Universal Robots PolyScope program: reciprocal_p1_3.urp

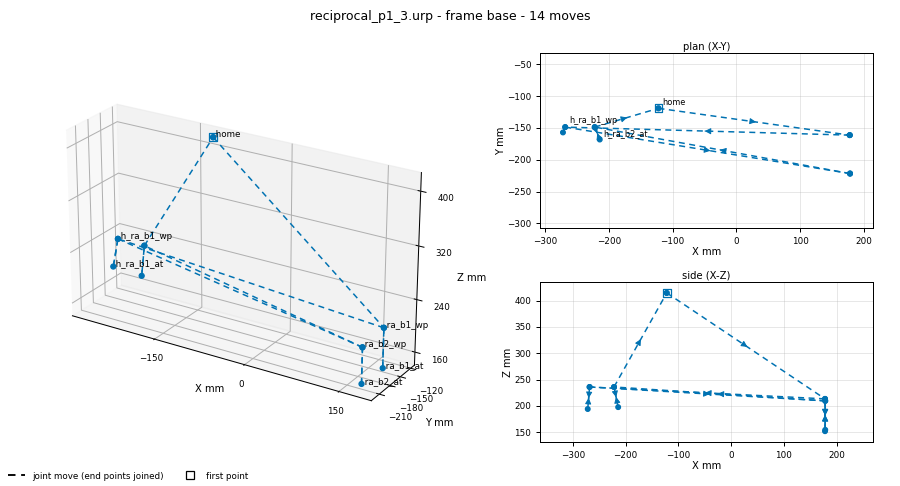
[picture p0: tool path of reciprocal_p1_3.urp in frame base, 14 of 14 moves have a stored position in this frame; points joined in program order, loops and branches not executed]
Program reciprocal_p1_3 (installation=default directory=/programs/usbdisk/ITER createdIn=5.3.1.64192 lastSavedIn=5.3.1.64192 robotSerialNumber=20195300365)
Calibrated DH parameters: a=[-0.000093, -0.190649, -0.212673, 0.000091, -0.000205, 0]; d=[0.151591, 44.061648, -42.488068, -1.442789, 0.085322, 0.091911]; alpha=[1.570082, -0.003447, 0.007513, 1.572293, -1.571904, 0]; deltaTheta=[0, -0.672656, 0.728185, -0.055522, 0.000005, 0]
Robot Program (runOnlyOnce=false)
  URCap Gripper Activate (Robotiq_Grippers, Robotiq Inc.) dataModel(ResetAndActivateKey=false)
  URCap Gripper (Robotiq_Grippers, Robotiq Inc.) dataModel(position=50.0, force=100.0, speed=100.0, positionInDouble=50.0, forceInDouble=100.0, speedInDouble=100.0, slaveIds=[9], blocking=true)
  MoveJ speed 60 deg/s, acceleration 80 deg/s^2 (useActiveTCP=true) feature=Base
    Waypoint home: TCP in base x=-122.15 y=-119.32 z=414.454 mm, rx=2.2563 ry=2.1459 rz=-0.0481 rad; joints [-85.681, -56.776, -79.802, -131.025, 89.944, -262.833] deg
  Folder Roof_A
    MoveJ speed 60 deg/s, acceleration 80 deg/s^2 (useActiveTCP=true) feature=Base
      Waypoint ra_b1_wp: TCP in base x=178.147 y=-161.416 z=213.493 mm, rx=2.2107 ry=2.1864 rz=-0.0129 rad; joints [-8.931, -69.528, -131.792, -67.419, 88.9, -187.899] deg
      Waypoint ra_b1_at: TCP in base x=178.14 y=-161.425 z=152.15 mm, rx=2.2108 ry=2.1863 rz=-0.013 rad; joints [-8.971, -81.208, -143.947, -43.587, 88.771, -187.8] deg
      URCap Gripper (Robotiq_Grippers, Robotiq Inc.) dataModel(position=100.0, force=100.0, speed=100.0, positionInDouble=100.0, forceInDouble=100.0, speedInDouble=100.0, slaveIds=[9], blocking=true)
      Waypoint ra_b1_wp: TCP in base x=178.147 y=-161.416 z=213.493 mm, rx=2.2107 ry=2.1864 rz=-0.0129 rad; joints [-8.931, -69.528, -131.792, -67.419, 88.9, -187.899] deg
      Waypoint h_ra_b1_wp: TCP in base x=-268.55 y=-148.787 z=236.04 mm, rx=2.7608 ry=-0.1306 rz=0.0749 rad; joints [-131.096, -88.368, -118.927, -47.1, 105.838, -213.026] deg
      Waypoint h_ra_b1_at: TCP in base x=-272.048 y=-157.193 z=194.251 mm, rx=2.7928 ry=-0.086 rz=0.1068 rad; joints [-130.55, -96.287, -122.586, -37.872, 105.802, -214.66] deg
      URCap Gripper (Robotiq_Grippers, Robotiq Inc.) dataModel(position=50.0, force=100.0, speed=100.0, positionInDouble=50.0, forceInDouble=100.0, speedInDouble=100.0, slaveIds=[9], blocking=true)
      Waypoint h_ra_b1_wp: TCP in base x=-268.55 y=-148.787 z=236.04 mm, rx=2.7608 ry=-0.1306 rz=0.0749 rad; joints [-131.096, -88.368, -118.927, -47.1, 105.838, -213.026] deg
    MoveJ speed 60 deg/s, acceleration 80 deg/s^2 (useActiveTCP=true) feature=Base
      Waypoint ra_b2_wp: TCP in base x=178.587 y=-221.707 z=209.682 mm, rx=2.2093 ry=2.1872 rz=-0.0611 rad; joints [-23.097, -83.646, -122.705, -62.748, 87.545, -202.118] deg
      Waypoint ra_b2_at: TCP in base x=178.563 y=-221.705 z=154.679 mm, rx=2.2094 ry=2.1872 rz=-0.0612 rad; joints [-23.123, -93.044, -131.897, -44.166, 87.443, -202.046] deg
      URCap Gripper (Robotiq_Grippers, Robotiq Inc.) dataModel(position=100.0, force=100.0, speed=100.0, positionInDouble=100.0, forceInDouble=100.0, speedInDouble=100.0, slaveIds=[9], blocking=true)
      Waypoint ra_b2_wp: TCP in base x=178.587 y=-221.707 z=209.682 mm, rx=2.2093 ry=2.1872 rz=-0.0611 rad; joints [-23.097, -83.646, -122.705, -62.748, 87.545, -202.118] deg
      Waypoint h_ra_b2_wp: TCP in base x=-222.173 y=-148.778 z=236.048 mm, rx=2.7617 ry=-0.0717 rz=0.0011 rad; joints [-121.367, -76.176, -130.557, -44.074, 100.878, -206.047] deg
      Waypoint h_ra_b2_at: TCP in base x=-214.314 y=-168.312 z=197.793 mm, rx=2.8721 ry=-0.0559 rz=-0.0607 rad; joints [-115.061, -82.329, -135.249, -37.27, 94.17, -201.737] deg
      URCap Gripper (Robotiq_Grippers, Robotiq Inc.) dataModel(position=50.0, force=100.0, speed=100.0, positionInDouble=50.0, forceInDouble=100.0, speedInDouble=100.0, slaveIds=[9], blocking=true)
      Waypoint h_ra_b2_wp: TCP in base x=-222.173 y=-148.778 z=236.048 mm, rx=2.7617 ry=-0.0717 rz=0.0011 rad; joints [-121.367, -76.176, -130.557, -44.074, 100.878, -206.047] deg
  MoveJ speed 60 deg/s, acceleration 80 deg/s^2 (useActiveTCP=true) feature=Base
    Waypoint home: TCP in base x=-122.15 y=-119.32 z=414.454 mm, rx=2.2563 ry=2.1459 rz=-0.0481 rad; joints [-85.681, -56.776, -79.802, -131.025, 89.944, -262.833] deg
